// TIA Portal V19 export
TYPE "LUC_typeSignalStackStateBehaviour"
TITLE = LUC_typeSignalStackStateBehavior
// Behavior settings for the signal stack - belonging to machine states
// stored: Access Published
   STRUCT
      static { ExternalWritable := 'False'} : "LUC_typeSignalStackByBool";
      flashing { ExternalWritable := 'False'} : "LUC_typeSignalStackByBool";
   END_STRUCT;
END_TYPE
